{attribute 'linkalways'} 
{attribute 'no_explicit_call' := 'This FB is a CLASS and must be accessed using methods or properties'}
{attribute 'enable_dynamic_creation'}
FUNCTION_BLOCK Node_F_VN_WarpAffine EXTENDS VisionNode
VAR
	ipSrcImage : _ITcVnImage;
    ipDestImage : _ITcVnImage;
    aTransformationMatrix : _TcVnMatrix2x3_LREAL;
    hrPrev : _HRESULT(S_OK);
	hresult : _HRESULT(S_OK);
END_VAR

METHOD PUBLIC  Clone : I_Node
VAR
	pNode : POINTER TO Node_F_VN_WarpAffine;
END_VAR
pNode := __NEW(Node_F_VN_WarpAffine);
Clone := pNode^;
END_METHOD

METHOD FB_init : BOOL
VAR_INPUT
	bInitRetains : BOOL; // if TRUE, the retain variables are initialized (warm start / cold start)
	bInCopyCode : BOOL;  // if TRUE, the instance afterwards gets moved into the copy code (online change)
END_VAR
AddInput('ipSrcImage', ipSrcImage);
AddInput('aTransformationMatrix', aTransformationMatrix);
AddInput('hrPrev', hrPrev);
AddOutput('ipDestImage', ipDestImage);
AddOutput('hresult',hresult);
END_METHOD

METHOD PROTECTED OnExecute
hresult.Value := F_VN_WarpAffine(
	ipSrcImage := ipSrcImage.Value, 
	ipDestImage := ipDestImage.Value, 
	aTransformationMatrix := aTransformationMatrix.Value, 
	hrPrev := hrPrev.Value);
END_METHOD

METHOD PUBLIC PreExecutionCheck
VAR_INPUT
	Check : I_PreExecutionChecks;
END_VAR
Check.IsTrue(ipSrcImage.IsValid, 'ipSrcImage must contain an image');
END_METHOD

END_FUNCTION_BLOCK

(* stored: Version 1.1.0.1, ProductVersion 3.1.4024.15
   POU Node_F_VN_WarpAffine: Id {f97904e4-baa6-0525-14ce-d1c40c66ae9d}, SpecialFunc None
   Folder Constructor: Id {61121522-004a-0dad-330a-895e0666bc78}
   Method Clone: Id {cb3e4ef3-72ad-0db4-02b2-6d1a5864c340}
   Method FB_init: Id {9ef70fb1-f9ce-05b3-1a69-25e20328dd4e}
   Method OnExecute: Id {6f32259f-6ce8-0596-0946-3c2e79a78f93}
   Method PreExecutionCheck: Id {0d24a3a7-6174-077c-324b-2d68d67139a4} *)
